PROGRAM MAIN2_RS485
VAR
	RS485_V2:ARRAY[1..4] OF FB_WarehouseSensorCtrl;
	
	i	: INT := 1;
	j	: INT;
	k	: INT;
	arr485sensor					: ARRAY [1..400] OF BOOL;

END_VAR

RS485_V2[1](bEnable:=TRUE);
RS485_V2[2](bEnable:=TRUE,UnitID := 2);
RS485_V2[3](bEnable:=TRUE,UnitID := 3);
RS485_V2[4](bEnable:=TRUE,UnitID := 4);

RS485_V2[1].ErrorId;
RS485_V2[2].ErrorId;
RS485_V2[3].ErrorId;
RS485_V2[4].ErrorId;

RS485_V2[1].RS485_ErrorCount;
RS485_V2[2].RS485_ErrorCount;
RS485_V2[3].RS485_ErrorCount;
RS485_V2[4].RS485_ErrorCount;

FOR i := 1 TO 400 DO
	k := i MOD 100;
	IF k = 0 THEN
		j := i/100;
		k := 100;
	ELSE
		j := (i/100) + 1;
	END_IF
	arr485sensor[i]:= RS485_V2[j].stRS485Controller.stSliderStatusALL.bPos[k];
END_FOR

END_PROGRAM

(* stored: Version 1.1.0.1, ProductVersion 3.1.4024.13
   POU MAIN2_RS485: Id {a5a8cde1-02dd-4659-8488-d46553febe67}, SpecialFunc None *)
